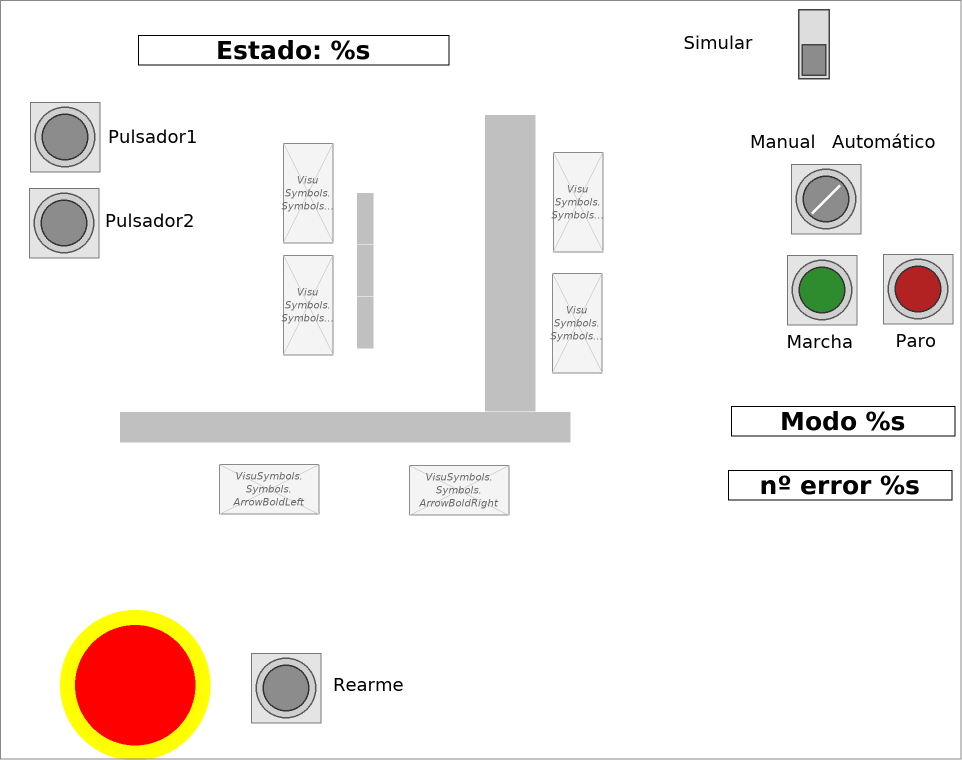
VISUALIZATION SimuladorPrensa  // 962x760
    PushSwitch (30,102 70x70), variable: IO.Pulsador1, behaviour: TAP, style: Switch-PushSwitch-Gray
    Rectangle (120,412 150x30), colour toggle: IO.SensorFora
        OnMouseClick: toggle IO.SensorFora
    Rectangle (270,412 150x30), colour toggle: Not IO.SensorFora and Not io.SensorDentro
    Rectangle (420,412 150x30), colour toggle: IO.SensorDentro
        OnMouseClick: toggle IO.SensorDentro
    Rectangle (357,193 16x51), colour toggle: IO.SensorAberto
        OnMouseClick: toggle IO.SensorAberto
    Rectangle (357,245 16x51), colour toggle: Not IO.SensorAberto and Not IO.SensorPechado
    Rectangle (357,297 16x51), colour toggle: IO.SensorPechado
        OnMouseClick: toggle IO.SensorPechado
    Rectangle (485,115 50x100), colour toggle: IO.SensorArriba
        OnMouseClick: toggle IO.SensorArriba
    Rectangle (485,214 50x100), colour toggle: Not io.SensorArriba and Not IO.SensorAbaixo
    Rectangle (485,311 50x100), colour toggle: IO.SensorAbaixo
        OnMouseClick: toggle IO.SensorAbaixo
    Rectangle (138,35 311x30), "Estado: %s", text variable: ModoAutomatico.EstadoPrensa
    Image (283,143 50x100), colour toggle: IO.ElectroAbrir, image: VisuSymbols.Symbols.ArrowBoldUp
        OnMouseDown: toggle IO.PulsadorAbrir
        OnMouseUp: toggle IO.PulsadorAbrir
    Image (283,255 50x100), colour toggle: IO.ElectroPechar, image: VisuSymbols.Symbols.ArrowBoldDown
        OnMouseDown: toggle IO.PulsadorPechar
        OnMouseUp: toggle IO.PulsadorPechar
    Image (553,152 50x100), colour toggle: IO.ElectroLiberar, image: VisuSymbols.Symbols.ArrowBoldUp
        OnMouseDown: toggle IO.PulsadorLiberar
        OnMouseUp: toggle IO.PulsadorLiberar
    Image (552,273 50x100), colour toggle: IO.ElectroPrensar, image: VisuSymbols.Symbols.ArrowBoldDown
        OnMouseDown: toggle IO.PulsadorPrensar
        OnMouseUp: toggle IO.PulsadorPrensar
    Image (409,465 100x50), colour toggle: IO.ElectroEntrar, image: VisuSymbols.Symbols.ArrowBoldRight
        OnMouseDown: toggle IO.PulsadorEntrar
        OnMouseUp: toggle IO.PulsadorEntrar
    Image (219,464 100x50), colour toggle: IO.ElectroSair, image: VisuSymbols.Symbols.ArrowBoldLeft
        OnMouseDown: toggle IO.PulsadorSair
        OnMouseUp: toggle IO.PulsadorSair
    Ellipse (60,610 150x150)
    Ellipse (75,625 120x120), colour toggle: Not IO.SafetyOK
        OnMouseClick: toggle IO.SafetyOK
    PushSwitch (251,653 70x70), variable: IO.ResetErrores, behaviour: TAP, style: Switch-PushSwitch-Gray
    RotarySwitch (791,164 70x70), variable: IO.ManualAuto, behaviour: TOGGLE, style: Switch-RotarySwitch-Gray
    PushSwitch (787,255 70x70), variable: IO.Marcha, behaviour: TAP, style: Switch-PushSwitch-Green
    Rectangle (731,406 224x30), "Modo %s", text variable: VariablesGlobales.ModoMaquina
    PushSwitch (883,254 70x70), variable: IO.Paro, behaviour: TOGGLE, style: Switch-PushSwitch-Red
    Label (327,663 83x44), "Rearme"
    Label (107,115 92x44), "Pulsador1"
    Label (741,120 204x44), "Manual Automático"
    Label (774,320 92x44), "Marcha"
    Label (870,319 92x44), "Paro"
    PushSwitch (29,188 70x70), variable: IO.Pulsador2, behaviour: TAP, style: Switch-PushSwitch-Gray
    Label (104,199 92x44), "Pulsador2"
    DipSwitch (779,9 70x70), variable: VariablesGlobales.Simular, behaviour: TOGGLE, style: Switch-DipSwitch-Gray
    Label (672,21 92x44), "Simular"
    Rectangle (728,470 224x30), "nº error %s", text variable: gesAlarmas.PrimeiroErro
END_VISUALIZATION

(* stored: Version 1.1.0.1, ProductVersion 3.1.4024.9
   Visu SimuladorPrensa: Id {2a67b6ba-c2ac-495f-bfb8-50dd27f52a32} *)
